// TIA Portal V16 export
// export: Created 2022-11-01T21:54:10.1418767Z, ExportSetting WithDefaults, DisplayName Totally Integrated Automation Portal, DisplayVersion V16, DisplayName TIA Portal Version Control Interface, DisplayVersion V16, DisplayName TIA Portal Openness, DisplayVersion V16, DisplayName SINAMICS Startdrive Advanced, DisplayVersion V16, DisplayName SINAMICS Startdrive G130, G150, S120, S150, SINAMICS MV, S210, DisplayVersion V16, DisplayName SINAMICS Startdrive G110M, G120, G120C, G120D, G120P, DisplayVersion V16, DisplayName STEP 7 Professional, DisplayVersion V16, DisplayName STEP 7 Safety, DisplayVersion V16, DisplayName WinCC Professional, DisplayVersion V16
VAR_GLOBAL   // PLC tag table "AI C900"
   iTIR901 AT %MW1700 : Int;
   iTIR902 AT %MW1702 : Int;
   iTIR903 AT %MW1704 : Int;
   iTIR904 AT %MW1706 : Int;
   iTIR905 AT %MW1708 : Int;
   iTIR906 AT %MW1710 : Int;
   iTIR907 AT %MW1712 : Int;
   iTIR908 AT %MW1714 : Int;
   iTIR909 AT %MW1716 : Int;
   iTIR910 AT %MW1718 : Int;
   iTIR911 AT %MW1720 : Int;
   iTIR912 AT %MW1722 : Int;
   iTIR913 AT %MW1724 : Int;
   iTIR914 AT %MW1726 : Int;
   iTIR915 AT %MW1728 : Int;
   iTIR916 AT %MW1730 : Int;
   iTIR917 AT %MW1732 : Int;
   iTIR918 AT %MW1734 : Int;
   iTIR919 AT %MW1736 : Int;
   iTIR920 AT %MW1738 : Int;
   iTIR921 AT %MW1740 : Int;
   iTIR922 AT %MW1742 : Int;
   iTIR923 AT %MW1744 : Int;
   iTIR924 AT %MW1746 : Int;
   iTIR925 AT %MW1748 : Int;
   iTIR926 AT %MW1750 : Int;
   iTIR927 AT %MW1752 : Int;
   iTIR928 AT %MW1754 : Int;
   iTIR929 AT %MW1756 : Int;
   iTIR930 AT %MW1758 : Int;
   iTIR931 AT %MW1760 : Int;
   iPIR901 AT %MW1762 : Int;
   iPIR902 AT %MW1764 : Int;
   iPIR903 AT %MW1766 : Int;
   iPIR904 AT %MW1768 : Int;
   iPIR905 AT %MW1770 : Int;
   iPIR906 AT %MW1772 : Int;
   iPIR907 AT %MW1774 : Int;
   iPIR908 AT %MW1776 : Int;
   iPIR909 AT %MW1778 : Int;
   iPIR910 AT %MW1780 : Int;
   iPIR911 AT %MW1782 : Int;
   iPIR912 AT %MW1784 : Int;
   iPIR913 AT %MW1786 : Int;
   iPIR914 AT %MW1788 : Int;
   iPIR915 AT %MW1790 : Int;
   iLIR900 AT %MW1792 : Int;
   iLIR901 AT %MW1794 : Int;
   iLIR902 AT %MW1796 : Int;
   iLIR903 AT %MW1798 : Int;
   iLIR904 AT %MW1800 : Int;
   iLIR905 AT %MW1802 : Int;
   iLIR906 AT %MW1804 : Int;
   iLIR907 AT %MW1806 : Int;
   iLIR908 AT %MW1808 : Int;
   iLIR909 AT %MW1810 : Int;
   iLIR910 AT %MW1812 : Int;
   iLIR911 AT %MW1814 : Int;
   iLIR912 AT %MW1816 : Int;
   iLIR913 AT %MW1818 : Int;
   iLIR914 AT %MW1820 : Int;
   iFIR901 AT %MW1822 : Int;
   iFIR902 AT %MW1824 : Int;
   iFIR903 AT %MW1826 : Int;
   iFIR904 AT %MW1828 : Int;
   iFIR905 AT %MW1830 : Int;
   iFIR906 AT %MW1832 : Int;
   iFIR907 AT %MW1834 : Int;
   iFIR908 AT %MW1836 : Int;
   iFIR909 AT %MW1838 : Int;
   iFIR910 AT %MW1840 : Int;
   iFIR911 AT %MW1842 : Int;
   iFIR912 AT %MW1844 : Int;
   iPIR916 AT %MW1866 : Int;
   iPIR917 AT %MW1868 : Int;
   iPIR918 AT %MW1870 : Int;
   iPIR919 AT %MW1872 : Int;
   iPIR920 AT %MW1874 : Int;
END_VAR
